FUNCTION_BLOCK FB_Torque_prediction_ST
VAR_INPUT
END_VAR
VAR_OUTPUT
END_VAR
VAR
	Lh_full: BOOL;
	Lh_half: BOOL;
	Equal: BOOL;
	Rh_half: BOOL;
	Rh_full: BOOL;
	
	Lh_full_selected: BOOL;
	Lh_half_selected: BOOL;
	Equal_selected: BOOL;
	Rh_half_selected: BOOL;
	Rh_full_selected: BOOL;
	
	R_TRIG0: R_TRIG;
	R_TRIG1: R_TRIG;
	R_TRIG2: R_TRIG;
	R_TRIG3: R_TRIG;
	R_TRIG4: R_TRIG;
END_VAR

R_TRIG0(CLK:= Torque_prediction.Lh_full_request, Q=> Lh_full_selected);
R_TRIG1(CLK:= Torque_prediction.Lh_half_request, Q=> Lh_half_selected);
R_TRIG2(CLK:= Torque_prediction.Equal_request, Q=> Equal_selected);
R_TRIG3(CLK:= Torque_prediction.Rh_half_request, Q=> Rh_half_selected);
R_TRIG4(CLK:= Torque_prediction.Rh_full_request, Q=> Rh_full_selected);

IF Lh_full_selected THEN
	Torque_prediction.Lh_full := 1;
	Torque_prediction.Lh_half := 0;
	Torque_prediction.Equal := 0;
	Torque_prediction.Rh_half := 0;
	Torque_prediction.Rh_full := 0;
ELSIF Lh_half_selected THEN
	Torque_prediction.Lh_full := 0;
	Torque_prediction.Lh_half := 1;
	Torque_prediction.Equal := 0;
	Torque_prediction.Rh_half := 0;
	Torque_prediction.Rh_full := 0;
ELSIF Equal_selected THEN
	Torque_prediction.Lh_full := 0;
	Torque_prediction.Lh_half := 0;
	Torque_prediction.Equal := 1;
	Torque_prediction.Rh_half := 0;
	Torque_prediction.Rh_full := 0;
ELSIF Rh_half_selected THEN
	Torque_prediction.Lh_full := 0;
	Torque_prediction.Lh_half := 0;
	Torque_prediction.Equal := 0;
	Torque_prediction.Rh_half := 1;
	Torque_prediction.Rh_full := 0;
ELSIF Rh_full_selected THEN
	Torque_prediction.Lh_full := 0;
	Torque_prediction.Lh_half := 0;
	Torque_prediction.Equal := 0;
	Torque_prediction.Rh_half := 0;
	Torque_prediction.Rh_full := 1;
END_IF

Torque_prediction.Lh_full_request := 0;
Torque_prediction.Lh_half_request := 0;
Torque_prediction.Equal_request := 0;
Torque_prediction.Rh_half_request := 0;
Torque_prediction.Rh_full_request := 0;

END_FUNCTION_BLOCK

(* stored: Version 1.1.0.1, ProductVersion 3.1.4024.0
   POU FB_Torque_prediction_ST: Id {121525ac-afdd-4a57-bdd6-f051485a00d4}, SpecialFunc None *)
